TYPE ST_Point :
STRUCT
    x : INT;
    y : INT;
END_STRUCT
END_TYPE

(* stored: Version 1.1.0.1
   DUT ST_Point: Id {51ad963e-cdac-4f9e-a988-9f01715b910e} *)
